FUNCTION_BLOCK FB_LamparaMemorizada_IL
VAR_INPUT
END_VAR
VAR_OUTPUT
END_VAR
VAR
    Lampara AT %Q*: BOOL;
    PulsadorConexion AT %I*: BOOL;
    PulsadorDesconexion AT %I*: BOOL;
END_VAR

// NETWORK 1
// instruction list
LD      PulsadorConexion
S       Lampara
LD      PulsadorDesconexion
R       Lampara

END_FUNCTION_BLOCK

(* stored: Version 1.1.0.1, ProductVersion 3.1.4024.15
   POU FB_LamparaMemorizada_IL: Id {cb55df0a-4d38-47ba-9d76-11d64b3ed990}, SpecialFunc None *)
